# EPICS SNL sequencer program: apps/waveformApp/src/waveform.st
/*
   N.Baltzell

   waveform.st

   Read list of PV names from a file, fill their values in a waveform,
   preserving ordering.  Allow for arbitrary number of PVs, limited by
   MAXLEN below and waveform record's .NELM, truncating if greater.

   {P}{R}wf       = waveform of PV values
   {P}{R}wfnames  = waveform of PV names
   {P}{R}period   = waveform update period in seconds
   {P}{R}filename = name of file from which to read PV names
   {P}{R}wflen    = number of PV names read from file
   {P}{R}msg      = sequencer status message
   {P}{R}sleep    = whether to use epicsThreadSleep instead of delay
*/

program waveform

// allow sequencer to start before all PVs connected:
option -c;

// make reentrant (required for multiple instances):
option +r;

// run in safe mode:
option +s;

#ifdef VXWORKS
%%#include <vxWorks.h>
%%#include <ioLib.h>
int inFile
#else
%%FILE* inFile;
#endif

#define MAXLEN  100000
float wfIn[MAXLEN];     assign wfIn to {};

#define NPVSTATIC 9
float wfOut[MAXLEN];    assign wfOut    to "{P}{R}wf";
float wfDelay;          assign wfDelay  to "{P}{R}period";
string wfNames[MAXLEN]; assign wfNames  to "{P}{R}wfnames";
string msg;             assign msg      to "{P}{R}msg";
string filename;        assign filename to "{P}{R}filename";
int wfLen;              assign wfLen    to "{P}{R}wflen";
int wfRecLen;           assign wfRecLen to "{P}{R}wf.NELM";
int doSleep;            assign doSleep  to "{P}{R}sleep";
int zero;               assign zero     to "{P}{R}zero";

monitor wfDelay;
monitor doSleep;

int ii;
int nPVs;
int isTruncated;
string stmp;
string stub;
string prefix;

ss waveform {

  state start {

    entry {
      wfLen=0;
      isTruncated=0;
      nPVs=NPVSTATIC;
      sprintf(stub,"seq waveform(%s%s)",macValueGet("P"),macValueGet("R"));
      sprintf(prefix,"%s%s",macValueGet("P"),macValueGet("R"));
    }

    when (pvConnectCount() < nPVs) {
      printf("\n%s - Waiting for Static PVs (%d/%d)\n",stub,pvConnectCount(),nPVs);
      sprintf(msg,"Waiting for Static PVs (%d/%d)",pvConnectCount(),nPVs);
      pvPut(msg);
      epicsThreadSleep(1);
    } state start

    when () {} state init

  }

  state init {

    when () {
      sprintf(msg,"Assigning PVs");
      pvPut(msg);
      pvPut(wfLen);
      pvGet(filename);
      pvGet(wfRecLen);
      if (wfRecLen > MAXLEN) {
        printf("%s - WARNING:  %swf.NELM is greater than sequencer's MAXLEN\n",stub,prefix);
      }
      sprintf(msg,"Opening file:  %s",filename);
      printf("%s - %s\n",stub,msg);
      pvPut(msg);
#ifdef VXWORKS
      inFile = open(filename,O_RDONLY);
#else
      inFile = fopen(filename,"r");
#endif
      if (!inFile) {
        sprintf(msg,"Error Reading %s",filename);
        pvPut(msg);
        printf("%s - %s\n",stub,msg);
      }
      else {
        while ((fscanf(inFile,"%s",stmp))==1) {
          if (wfLen >= wfRecLen || wfLen >= MAXLEN) {
            sprintf(msg,"#PVs > NELM/MAXLEN.  Truncating.");
            pvPut(msg);
            printf("%s - %s\n",stub,msg);
            isTruncated=1;
            break;
          }
          if (stmp[0] == '#') {
              pvAssign(wfIn[wfLen],"{P}{R}zero");
              nPVs -= 1;
          }
          else {
              pvAssign(wfIn[wfLen],stmp);
          }
          pvMonitor(wfIn[wfLen]);
          sprintf(wfNames[wfLen],"%s",stmp);
          wfLen++;
        }
        fclose(inFile);
      }
      pvPut(wfLen);
      pvPut(wfNames);
      nPVs += wfLen;
    } state wait

  }

  state wait {

    when (wfLen <= 0) {
      sprintf(msg,"Zero PVs Read from %s",filename);
      pvPut(msg);
      printf("%s - %s - EXITING SEQUENCER\n",stub,msg);
    } exit

    when (pvConnectCount() < nPVs) {
      sprintf(msg,"Waiting for PVs (%d/%d)",pvConnectCount(),nPVs);
      pvPut(msg);
      printf("%s - %s\n",stub,msg);
      epicsThreadSleep(1);
    } state wait

    when () {} state run
  }

  state run {

    entry {
      if (isTruncated) sprintf(msg,"OK - Running Truncated");
      else             sprintf(msg,"OK - Running");
      pvPut(msg);
      printf("%s - %s\n",stub,msg);
    }

    when (pvConnectCount() < nPVs) {} state wait

    when (doSleep || delay(wfDelay)) {
      if (doSleep) epicsThreadSleep(wfDelay);
      for (ii=0; ii<wfLen; ii++) wfOut[ii]=wfIn[ii];
      pvPut(wfOut);
    } state run

  }

}
